{attribute addProperty BoxType "EK1100-0000-0018"}
{attribute addProperty Id "Beckhoff_EL47xxEK1122Beckhoff_EL47xxEK1122_4AFA0311162A_0001_EL4712_0000_0000EL4712_AF3811B143354.125A_0002_EL4712_0000_0001EL4712_AF3811B143354.125A_0003_EL4732_0001_0000EL4732_A4B0F6DE12916.125A_0004_EL4732_0000_0002EL4732_AF3811B143354.125A_0005_EL4732_0000_0003EL4732_AF3811B143354.125A_0006_EL4732_0000_0004EL4732_AF3811B143354.125"}
{attribute addProperty CRC "2522763668"}
{attribute addProperty SizeInBites "2310"}
{attribute addProperty SizeInBytes "288.75"}
TYPE Beckhoff_EL47xx_965E5194 EXTENDS EK1100_179A0949 :
STRUCT
	{attribute addProperty Name "Beckhoff_EL47xxEK1122"}
	Beckhoff_EL47xxEK1122 : Beckhoff_EL47xxEK1122_4AFA0311;
	{attribute addProperty Name "A_0001_EL4712_0000_0000"}
	A_0001_EL4712_0000_0000 : EL4712_AF3811B1;
	{attribute addProperty Name "A_0002_EL4712_0000_0001"}
	A_0002_EL4712_0000_0001 : EL4712_AF3811B1;
	{attribute addProperty Name "A_0003_EL4732_0001_0000"}
	A_0003_EL4732_0001_0000 : EL4732_A4B0F6DE;
	{attribute addProperty Name "A_0004_EL4732_0000_0002"}
	A_0004_EL4732_0000_0002 : EL4732_AF3811B1;
	{attribute addProperty Name "A_0005_EL4732_0000_0003"}
	A_0005_EL4732_0000_0003 : EL4732_AF3811B1;
	{attribute addProperty Name "A_0006_EL4732_0000_0004"}
	A_0006_EL4732_0000_0004 : EL4732_AF3811B1;
END_STRUCT
END_TYPE

(* stored: Version 1.2.0.0, ProductVersion 3.1.4024.9
   DUT Beckhoff_EL47xx_965E5194: Id {443dfde7-44dc-4dba-be56-902b91bcc4bc} *)
